FUNCTION_BLOCK Test_StringSplitter_Handles_Empty_String EXTENDS TUnitTestBase
VAR
END_VAR

METHOD  Execute
VAR_INST
    StringSplitter : TStringSplitter;
END_VAR
Test_Started();

StringSplitter.Init(
    Str    := '',
    Delim1 := '$T',
    Delim2 := '');

AssertEquals_STRING(
    Expected := '',
    Actual   := StringSplitter.GetNext(),
    VariableName  := 'StringSplitter.GetNext()');

AssertEquals_BOOL(
    Expected := FALSE,
    Actual   := StringSplitter.HasMore(),
    VariableName  := 'StringSplitter.HasMore()');


Test_Finished();
END_METHOD

END_FUNCTION_BLOCK

(* stored: Version 1.1.0.1, ProductVersion 3.1.4024.3
   POU Test_StringSplitter_Handles_Empty_String: Id {3a7cf2cc-79a9-0132-02fd-8eb652eaae4e}, SpecialFunc None
   Method Execute: Id {a479ed32-d15a-0b5d-0a09-99fd0530190f} *)
